SUBAPPLICATION AR_HZ_TO_Q_Publish_OPC (* Remote-Hz-Subscribe -> feste Skalierung -> VT-Anzeige (Q_NumericValue_PHYSA) UND per OPC-UA publiziert (AR_PUBLISH_1). Buendelt AR_SUBSCRIBE_1+initval_AR+AR_MUL_2+AR_TO_Q_Publish_OPC - ein Baustein je Puls-Geschwindigkeits-/Drehzahlsensor (Aufnahme B03, Igelband1/2 B10/B11, Saegeblatt B08), nur Parameter unterscheiden sich. *)
  (* Standard: 61499-2; Description: Copyright (c) 2026 Meisterschulen am Ostbahnhof This program and the accompanying materials are made available under the terms of the Eclipse Public License 2.0 which is available at https://www.eclipse.org/legal/epl-2.0/ SPDX-License-Identifier: EPL-2.0 *)
  (* Version 1.0, 2026-09-13, Franz Höpfinger, Meisterschulen am Ostbahnhof, initial implementation - herausgeloest aus Inputs_STG1.SUB (Aufnahme/Igelband1/Igelband2/Saegeblatt waren 4x nahezu identische AR_SUBSCRIBE_1+initval_AR+AR_MUL_2+AR_TO_Q_Publish_OPC-Ketten, nur Parameter unterschiedlich). *)
  (* Version 1.1, 2026-09-22, Franz Höpfinger, Meisterschulen am Ostbahnhof, Neuer optionaler Plug HZ_RAW_OUT (AR_SPLIT_2 vor AR_MUL eingefuegt) - Spiegel des noch unskalierten Rohwerts (Hz), fuer eine Diagnose-Anzeige (z.B. IO-Diagnose-Zeile), ohne einen zweiten eigenstaendigen Remote-Subscribe desselben Knotens zu brauchen (FORTE: 'Cannot add another one' bei doppeltem Self-Subscribe). Unverdrahtet lassen, wenn nicht gebraucht. *)
  PACKAGE MyLib::sys;
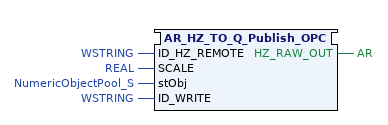
  VAR_INPUT
    ID_HZ_REMOTE : WSTRING; (* Remote-Subscribe-Adresse der publizierten Frequenz (Hz), z.B. FBs::Ventilsteuerung::Ventilsteuerung_STG1::RemoteSubStrings::AUFNAHME_GESCHWINDIGKEIT_HZ_REMOTE *)
    SCALE : REAL; (* Skalierungsfaktor Hz -> physikalische Einheit (z.B. 3.6/53 fuer km/h, 60.0 fuer U/min bei 1 Impuls/Umdrehung) *)
    stObj : logiBUS::utils::conversion::phys::NumericObjectPool_S; (* Object pool properties der VT-Zahlenvariable (u16ObjId, scale, offset, decimals) - z.B. FBs::const::DefaultPool_Numeric::NumberVariable_X_N *)
    ID_WRITE : WSTRING; (* Lokale Publish-Adresse (REAL, physikalischer Wert) - Web-Mirror/Dashboard/Self-Subscribe *)
  END_VAR
  PLUGS
    HZ_RAW_OUT : adapter::types::unidirectional::AR; (* Optional: Nur-Lese-Spiegel des noch unskalierten Rohwerts (Hz) vor der SCALE-Multiplikation, fuer weitere lokale Konsumenten (z.B. Diagnose-Anzeige) statt eigenem Remote-Subscribe. Unverdrahtet lassen, wenn nicht gebraucht. *)
  END_PLUGS
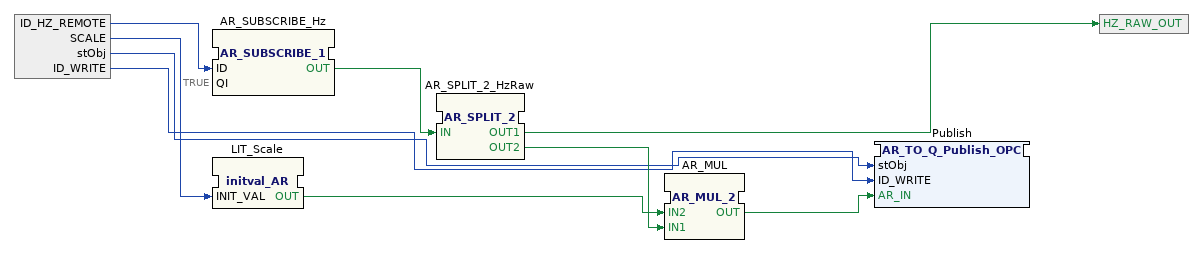
  FBS
    AR_SUBSCRIBE_Hz : adapter::net::AR_SUBSCRIBE_1(QI := TRUE);
    LIT_Scale : adapter::types::unidirectional::AR::initval::initval_AR;
    AR_SPLIT_2_HzRaw : adapter::events::unidirectional::AR_SPLIT_2;
    AR_MUL : adapter::iec61131::arithmetic::AR_MUL_2;
  END_FBS
  SUBAPPS
    Publish : MyLib::sys::AR_TO_Q_Publish_OPC;
  END_SUBAPPS
  DATA_CONNECTIONS
    ID_HZ_REMOTE TO AR_SUBSCRIBE_Hz.ID;
    SCALE TO LIT_Scale.INIT_VAL;
    stObj TO Publish.stObj;
    ID_WRITE TO Publish.ID_WRITE;
  END_CONNECTIONS
  ADAPTER_CONNECTIONS
    AR_SUBSCRIBE_Hz.OUT TO AR_SPLIT_2_HzRaw.IN;
    AR_SPLIT_2_HzRaw.OUT1 TO HZ_RAW_OUT;
    LIT_Scale.OUT TO AR_MUL.IN2;
    AR_MUL.OUT TO Publish.AR_IN;
    AR_SPLIT_2_HzRaw.OUT2 TO AR_MUL.IN1;
  END_CONNECTIONS
END_SUBAPPLICATION
